TYPE ST_GenericError EXTENDS ST_Error :
STRUCT
	Code	: DINT;
	Message	: Tc2_System.T_MaxString;
END_STRUCT
END_TYPE

(* stored: Version 1.1.0.1, ProductVersion 3.1.4024.14
   DUT ST_GenericError: Id {49ae69fd-0251-0b91-3d6c-84dfea2ea8b1} *)
